FUNCTION_BLOCK FillerCPM_Current
VAR_INPUT
	Filler_PulseInput : BOOL;
END_VAR
VAR_OUTPUT
	Current_Can_Pulses : REAL;
    CPM_Reading : REAL;
END_VAR
VAR
	fb_RisingEdge : R_TRIG;
    fb_MinuteTimer : TON;
    udiCurrentPulseCount : REAL := 0;
END_VAR

// Rising edge detection for pulse input
    fb_RisingEdge(CLK := Filler_PulseInput);
	IF fb_RisingEdge.Q THEN
        udiCurrentPulseCount := udiCurrentPulseCount + 1;
    END_IF
	// Minute timer
    fb_MinuteTimer(IN := TRUE, PT := T#20S); // Start timer automatically

    // When the minute timer expires
    IF fb_MinuteTimer.Q THEN
		
        // Store the current count as the last minute's count
        CPM_Reading := (udiCurrentPulseCount*3 * 0.75);
        // Reset the current pulse count for the new minute
        udiCurrentPulseCount := 0;
        // Reset the timer to start counting for the next minute
        fb_MinuteTimer(IN := FALSE); // Reset timer
        fb_MinuteTimer(IN := TRUE, PT := T#20S);//Restart timer
    END_IF

    // Output the current minute's pulse count
    Current_Can_Pulses := udiCurrentPulseCount;

END_FUNCTION_BLOCK

(* stored: Version 1.1.0.1, ProductVersion 3.1.4024.15
   POU FillerCPM_Current: Id {d39bcf92-5f78-4c9b-89a7-e98574a1fb4a}, SpecialFunc None *)
